// TIA Portal V19 export
FUNCTION "FC901_SafetyInputs" : Void   // FC901, F_LAD
{ S7_Optimized_Access := 'TRUE' }
// stored: AutoNumber false
BEGIN

REGION Network 1: Emergency stop on main cabinet
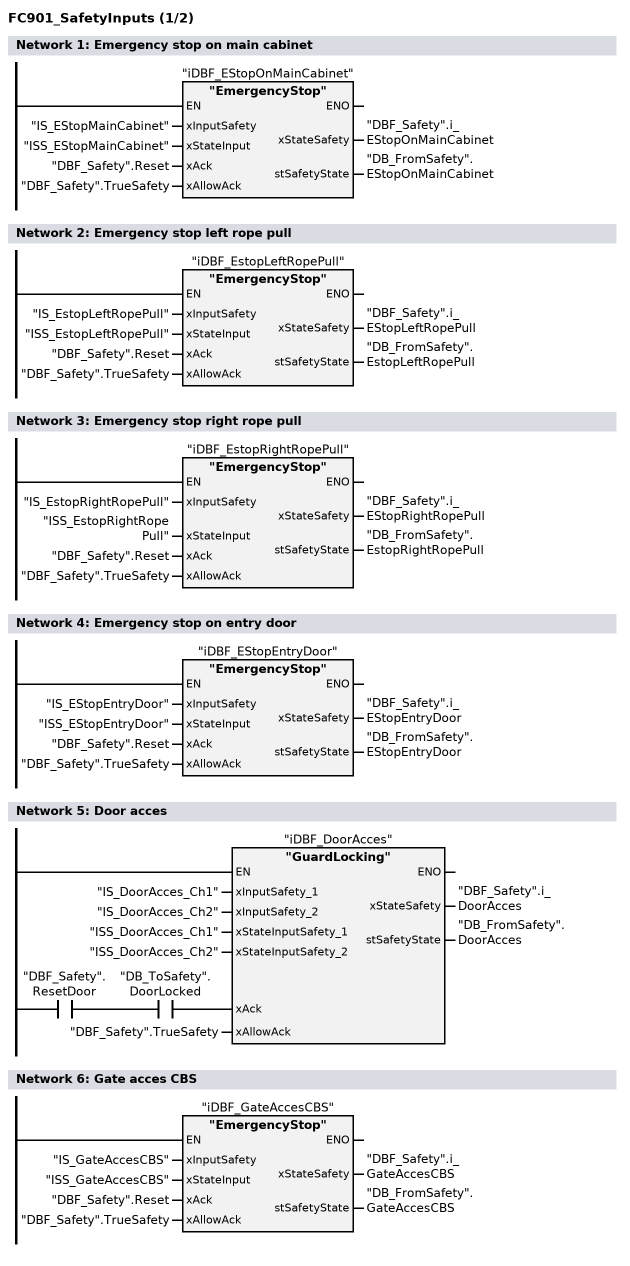
   RUNG wire#powerrail
      "iDBF_EStopOnMainCabinet"(xInputSafety := "IS_EStopMainCabinet", xStateInput := "ISS_EStopMainCabinet", xAck := "DBF_Safety".Reset, xAllowAck := "DBF_Safety".TrueSafety, xStateSafety => "DBF_Safety".i_EStopOnMainCabinet, stSafetyState => "DB_FromSafety".EStopOnMainCabinet)
   END_RUNG
   // the same network as SCL:
   "iDBF_EStopOnMainCabinet"(xInputSafety := "IS_EStopMainCabinet",   // "EmergencyStop"
                           xStateInput := "ISS_EStopMainCabinet",
                           xAck := "DBF_Safety".Reset,
                           xAllowAck := "DBF_Safety".TrueSafety,
                           xStateSafety => "DBF_Safety".i_EStopOnMainCabinet,
                           stSafetyState => "DB_FromSafety".EStopOnMainCabinet);
END_REGION

REGION Network 2: Emergency stop left rope pull
   RUNG wire#powerrail
      "iDBF_EstopLeftRopePull"(xInputSafety := "IS_EstopLeftRopePull", xStateInput := "ISS_EstopLeftRopePull", xAck := "DBF_Safety".Reset, xAllowAck := "DBF_Safety".TrueSafety, xStateSafety => "DBF_Safety".i_EStopLeftRopePull, stSafetyState => "DB_FromSafety".EstopLeftRopePull)
   END_RUNG
   // the same network as SCL:
   "iDBF_EstopLeftRopePull"(xInputSafety := "IS_EstopLeftRopePull",   // "EmergencyStop"
                           xStateInput := "ISS_EstopLeftRopePull",
                           xAck := "DBF_Safety".Reset,
                           xAllowAck := "DBF_Safety".TrueSafety,
                           xStateSafety => "DBF_Safety".i_EStopLeftRopePull,
                           stSafetyState => "DB_FromSafety".EstopLeftRopePull);
END_REGION

REGION Network 3: Emergency stop right rope pull
   RUNG wire#powerrail
      "iDBF_EstopRightRopePull"(xInputSafety := "IS_EstopRightRopePull", xStateInput := "ISS_EstopRightRopePull", xAck := "DBF_Safety".Reset, xAllowAck := "DBF_Safety".TrueSafety, xStateSafety => "DBF_Safety".i_EStopRightRopePull, stSafetyState => "DB_FromSafety".EstopRightRopePull)
   END_RUNG
   // the same network as SCL:
   "iDBF_EstopRightRopePull"(xInputSafety := "IS_EstopRightRopePull",   // "EmergencyStop"
                           xStateInput := "ISS_EstopRightRopePull",
                           xAck := "DBF_Safety".Reset,
                           xAllowAck := "DBF_Safety".TrueSafety,
                           xStateSafety => "DBF_Safety".i_EStopRightRopePull,
                           stSafetyState => "DB_FromSafety".EstopRightRopePull);
END_REGION

REGION Network 4: Emergency stop on entry door
   RUNG wire#powerrail
      "iDBF_EStopEntryDoor"(xInputSafety := "IS_EStopEntryDoor", xStateInput := "ISS_EStopEntryDoor", xAck := "DBF_Safety".Reset, xAllowAck := "DBF_Safety".TrueSafety, xStateSafety => "DBF_Safety".i_EStopEntryDoor, stSafetyState => "DB_FromSafety".EStopEntryDoor)
   END_RUNG
   // the same network as SCL:
   "iDBF_EStopEntryDoor"(xInputSafety := "IS_EStopEntryDoor",   // "EmergencyStop"
                         xStateInput := "ISS_EStopEntryDoor",
                         xAck := "DBF_Safety".Reset,
                         xAllowAck := "DBF_Safety".TrueSafety,
                         xStateSafety => "DBF_Safety".i_EStopEntryDoor,
                         stSafetyState => "DB_FromSafety".EStopEntryDoor);
END_REGION

REGION Network 5: Door acces
   RUNG wire#powerrail
      "iDBF_DoorAcces"(xAck := wire#w1, xInputSafety_1 := "IS_DoorAcces_Ch1", xInputSafety_2 := "IS_DoorAcces_Ch2", xStateInputSafety_1 := "ISS_DoorAcces_Ch1", xStateInputSafety_2 := "ISS_DoorAcces_Ch2", xAllowAck := "DBF_Safety".TrueSafety, xStateSafety => "DBF_Safety".i_DoorAcces, stSafetyState => "DB_FromSafety".DoorAcces)
   END_RUNG
   RUNG wire#powerrail
      Contact( "DBF_Safety".ResetDoor )
      Contact( "DB_ToSafety".DoorLocked )
   END_RUNG wire#w1
   // the same network as SCL:
   "iDBF_DoorAcces"(xInputSafety_1 := "IS_DoorAcces_Ch1",   // "GuardLocking"
                    xInputSafety_2 := "IS_DoorAcces_Ch2",
                    xStateInputSafety_1 := "ISS_DoorAcces_Ch1",
                    xStateInputSafety_2 := "ISS_DoorAcces_Ch2",
                    xAck := "DBF_Safety".ResetDoor AND "DB_ToSafety".DoorLocked,
                    xAllowAck := "DBF_Safety".TrueSafety,
                    xStateSafety => "DBF_Safety".i_DoorAcces,
                    stSafetyState => "DB_FromSafety".DoorAcces);
END_REGION

REGION Network 6: Gate acces CBS
   RUNG wire#powerrail
      "iDBF_GateAccesCBS"(xInputSafety := "IS_GateAccesCBS", xStateInput := "ISS_GateAccesCBS", xAck := "DBF_Safety".Reset, xAllowAck := "DBF_Safety".TrueSafety, xStateSafety => "DBF_Safety".i_GateAccesCBS, stSafetyState => "DB_FromSafety".GateAccesCBS)
   END_RUNG
   // the same network as SCL:
   "iDBF_GateAccesCBS"(xInputSafety := "IS_GateAccesCBS",   // "EmergencyStop"
                       xStateInput := "ISS_GateAccesCBS",
                       xAck := "DBF_Safety".Reset,
                       xAllowAck := "DBF_Safety".TrueSafety,
                       xStateSafety => "DBF_Safety".i_GateAccesCBS,
                       stSafetyState => "DB_FromSafety".GateAccesCBS);
END_REGION

REGION Network 7: Emergency stop in the control room
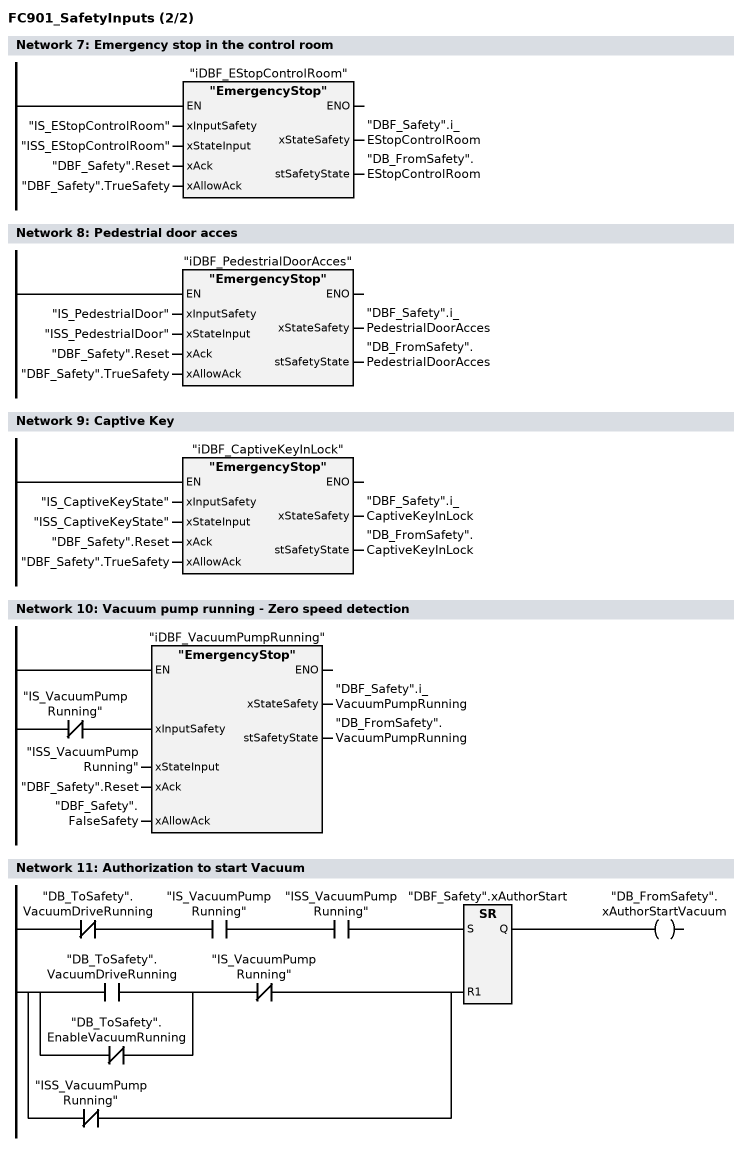
   RUNG wire#powerrail
      "iDBF_EStopControlRoom"(xInputSafety := "IS_EStopControlRoom", xStateInput := "ISS_EStopControlRoom", xAck := "DBF_Safety".Reset, xAllowAck := "DBF_Safety".TrueSafety, xStateSafety => "DBF_Safety".i_EStopControlRoom, stSafetyState => "DB_FromSafety".EStopControlRoom)
   END_RUNG
   // the same network as SCL:
   "iDBF_EStopControlRoom"(xInputSafety := "IS_EStopControlRoom",   // "EmergencyStop"
                           xStateInput := "ISS_EStopControlRoom",
                           xAck := "DBF_Safety".Reset,
                           xAllowAck := "DBF_Safety".TrueSafety,
                           xStateSafety => "DBF_Safety".i_EStopControlRoom,
                           stSafetyState => "DB_FromSafety".EStopControlRoom);
END_REGION

REGION Network 8: Pedestrial door acces
   RUNG wire#powerrail
      "iDBF_PedestrialDoorAcces"(xInputSafety := "IS_PedestrialDoor", xStateInput := "ISS_PedestrialDoor", xAck := "DBF_Safety".Reset, xAllowAck := "DBF_Safety".TrueSafety, xStateSafety => "DBF_Safety".i_PedestrialDoorAcces, stSafetyState => "DB_FromSafety".PedestrialDoorAcces)
   END_RUNG
   // the same network as SCL:
   "iDBF_PedestrialDoorAcces"(xInputSafety := "IS_PedestrialDoor",   // "EmergencyStop"
                           xStateInput := "ISS_PedestrialDoor",
                           xAck := "DBF_Safety".Reset,
                           xAllowAck := "DBF_Safety".TrueSafety,
                           xStateSafety => "DBF_Safety".i_PedestrialDoorAcces,
                           stSafetyState => "DB_FromSafety".PedestrialDoorAcces);
END_REGION

REGION Network 9: Captive Key
   RUNG wire#powerrail
      "iDBF_CaptiveKeyInLock"(xInputSafety := "IS_CaptiveKeyState", xStateInput := "ISS_CaptiveKeyState", xAck := "DBF_Safety".Reset, xAllowAck := "DBF_Safety".TrueSafety, xStateSafety => "DBF_Safety".i_CaptiveKeyInLock, stSafetyState => "DB_FromSafety".CaptiveKeyInLock)
   END_RUNG
   // the same network as SCL:
   "iDBF_CaptiveKeyInLock"(xInputSafety := "IS_CaptiveKeyState",   // "EmergencyStop"
                           xStateInput := "ISS_CaptiveKeyState",
                           xAck := "DBF_Safety".Reset,
                           xAllowAck := "DBF_Safety".TrueSafety,
                           xStateSafety => "DBF_Safety".i_CaptiveKeyInLock,
                           stSafetyState => "DB_FromSafety".CaptiveKeyInLock);
END_REGION

REGION Network 10: Vacuum pump running - Zero speed detection
   RUNG wire#powerrail
      "iDBF_VacuumPumpRunning"(xInputSafety := wire#w1, xStateInput := "ISS_VacuumPumpRunning", xAck := "DBF_Safety".Reset, xAllowAck := "DBF_Safety".FalseSafety, xStateSafety => "DBF_Safety".i_VacuumPumpRunning, stSafetyState => "DB_FromSafety".VacuumPumpRunning)
   END_RUNG
   RUNG wire#powerrail
      I_Contact( "IS_VacuumPumpRunning" )
   END_RUNG wire#w1
   // the same network as SCL:
   "iDBF_VacuumPumpRunning"(xInputSafety := NOT "IS_VacuumPumpRunning",   // "EmergencyStop"
                           xStateInput := "ISS_VacuumPumpRunning",
                           xAck := "DBF_Safety".Reset,
                           xAllowAck := "DBF_Safety".FalseSafety,
                           xStateSafety => "DBF_Safety".i_VacuumPumpRunning,
                           stSafetyState => "DB_FromSafety".VacuumPumpRunning);
END_REGION

REGION Network 11: Authorization to start Vacuum
   RUNG wire#powerrail
      I_Contact( "DB_ToSafety".VacuumDriveRunning )
      Contact( "IS_VacuumPumpRunning" )
      Contact( "ISS_VacuumPumpRunning" )
      S_SR(operand := "DBF_Safety".xAuthorStart, r1 := wire#w2)
      Coil( "DB_FromSafety".xAuthorStartVacuum )
   END_RUNG
   RUNG wire#powerrail
      Contact( "DB_ToSafety".VacuumDriveRunning )
      wire#w1
      I_Contact( "IS_VacuumPumpRunning" )
   END_RUNG wire#w2
   RUNG wire#powerrail
      I_Contact( "DB_ToSafety".EnableVacuumRunning )
   END_RUNG wire#w1
   RUNG wire#powerrail
      I_Contact( "ISS_VacuumPumpRunning" )
   END_RUNG wire#w2
   // the same network as SCL:
   IF NOT "DB_ToSafety".VacuumDriveRunning AND "IS_VacuumPumpRunning" AND "ISS_VacuumPumpRunning" THEN
       "DBF_Safety".xAuthorStart := TRUE;   // SR flip-flop
   END_IF;
   IF (("DB_ToSafety".VacuumDriveRunning OR NOT "DB_ToSafety".EnableVacuumRunning) AND NOT "IS_VacuumPumpRunning") OR NOT "ISS_VacuumPumpRunning" THEN
       "DBF_Safety".xAuthorStart := FALSE;
   END_IF;
   "DB_FromSafety".xAuthorStartVacuum := "DBF_Safety".xAuthorStart;
END_REGION
END_FUNCTION
